TYPE ST_Inputs :
STRUCT
	GRIP_CLOSED    			: BOOL;
	JOINT_FEEDBACK_SIGNAL	: ARRAY [1..GVL_RobotArmConstants.MAX_NUMBER_OF_JOINTS] OF ST_JointDirection;
END_STRUCT
END_TYPE

(* stored: Version 1.1.0.1, ProductVersion 3.1.4024.9
   DUT ST_Inputs: Id {d8030c2b-0c85-4476-bc48-afcf06e17b20} *)
